Fanuc KAREL source: kt00716.KL

-- PROVISIONAL review KL for V1013-1; original PC SHA256 591b56fd6934bd955fa81744cb0b58ec53032d090f19cc94bcf89cde4130fa38
-- Incomplete behavior may be omitted. Consult companion uncertainty JSON. Do not deploy.
PROGRAM KT00716
%NOLOCKGROUP
VAR
  OUT : BOOLEAN
-- UNRESOLVED_DECL H1 type=002017
-- UNRESOLVED_DECL H2 type=002017
BEGIN
  -- UNRESOLVED_PC offsets 5-19; opcodes 2E,22,9D,33,B4
  -- UNRESOLVED_PC offsets 24-38; opcodes 2E,22,9D,33,B4
  -- UNRESOLVED_PC offsets 43-57; opcodes 2E,22,9D,33,B4
  -- UNRESOLVED_PC offsets 62-76; opcodes 2E,22,9D,33,B4
  -- UNRESOLVED_PC offsets 81-98; opcodes 22,9D,33,63,23
  -- UNRESOLVED_PC offsets 103-107; opcodes 7F
END KT00716
